(* IEC 61131-3 sources: plc_generation_empirical_study/datasets/task_bank_v0_3_1/tasks/C08_B09_composite/negative_control, 1 file *)

(* ---- NC1.st ---- *)
FUNCTION_BLOCK C08_B09_composite
VAR_INPUT
    A_ItemPresent : BOOL;
    A_RejectClass : BOOL;
    A_TransferDone : BOOL;
    A_Reset : BOOL;
    B_Start : BOOL;
    B_Advance : BOOL;
    B_Pause : BOOL;
    B_Resume : BOOL;
    B_Abort : BOOL;
    B_Reset : BOOL;
    SubsystemBEnable : BOOL;
    CrossReset : BOOL;
END_VAR
VAR_OUTPUT
    A_Inspect : BOOL;
    A_AcceptGate : BOOL;
    A_RejectGate : BOOL;
    A_State : INT;
    B_Step1 : BOOL;
    B_Step2 : BOOL;
    B_Paused : BOOL;
    B_Aborted : BOOL;
    B_State : INT;
    CrossReady : BOOL;
    CrossBlocked : BOOL;
END_VAR

IF A_Reset THEN
    A_State := 0;
ELSE
    CASE A_State OF
        0: IF A_ItemPresent THEN A_State := 1; END_IF;
        1: IF A_RejectClass THEN A_State := 3; ELSE A_State := 2; END_IF;
        2: IF A_TransferDone THEN A_State := 0; END_IF;
        3: IF A_TransferDone THEN A_State := 0; END_IF;
        ELSE A_State := 0;
    END_CASE;
END_IF;
A_Inspect := A_State = 1;
A_AcceptGate := A_State = 2;
A_RejectGate := A_State = 3;

IF CrossReset THEN
    CrossReady := FALSE;
ELSIF A_Inspect THEN
    CrossReady := TRUE;
END_IF;
CrossBlocked := FALSE;

IF SubsystemBEnable AND CrossReady THEN
    IF B_Abort THEN
        B_State := 0;
        B_Paused := FALSE;
        B_Aborted := TRUE;
    ELSIF B_Reset AND (NOT B_Start) AND (NOT B_Advance) AND (NOT B_Pause) AND (NOT B_Resume) THEN
        B_Aborted := FALSE;
    ELSIF NOT B_Aborted THEN
        IF B_Pause AND ((B_State = 1) OR (B_State = 2)) THEN
            B_Paused := TRUE;
        ELSIF B_Resume THEN
            B_Paused := FALSE;
        END_IF;
        IF NOT B_Paused THEN
            CASE B_State OF
                0: IF B_Start THEN B_State := 1; END_IF;
                1: IF B_Advance THEN B_State := 2; END_IF;
                2: IF B_Advance THEN B_State := 3; END_IF;
                3: B_State := 3;
                ELSE B_State := 0;
            END_CASE;
        END_IF;
    END_IF;
    B_Step1 := (B_State = 1) AND (NOT B_Paused) AND (NOT B_Aborted);
    B_Step2 := (B_State = 2) AND (NOT B_Paused) AND (NOT B_Aborted);
ELSE
    B_Step1 := FALSE;
    B_Step2 := FALSE;
    B_Paused := FALSE;
    B_Aborted := FALSE;
    B_State := 0;
END_IF;

END_FUNCTION_BLOCK
